FUNCTION_BLOCK AI_ChannelStatus
VAR
	{attribute addProperty Name  "<#Under Range#>"}
	UnderRange AT %I* : BIT;
	{attribute addProperty Name  "<#Over Range#>"}
	OverRange AT %I* : BIT;
	{attribute addProperty Name  "<#Value greater then limit 1#>"}
	Limit_1_Greater AT %I* : BIT;
	{attribute addProperty Name  "<#Value smaller then limit 1#>"}
	Limit_1_Smaller AT %I* : BIT;
	{attribute addProperty Name  "<#Value greater then limit 2#>"}
	Limit_2_Greater AT %I* : BIT;
	{attribute addProperty Name  "<#Value smaller then limit 2#>"}
	Limit_2_Smaller AT %I* : BIT;
	{attribute addProperty Name  "<#Error"}
	Error AT %I* : BIT;
	{attribute 'hide'}
	Reserved_1_7 AT %I* : BIT;
	{attribute 'hide'}
	Reserved_2_0 AT %I* : BIT;
	{attribute 'hide'}
	Reserved_2_1 AT %I* : BIT;
	{attribute 'hide'}
	Reserved_2_2 AT %I* : BIT;
	{attribute 'hide'}
	Reserved_2_3 AT %I* : BIT;
	{attribute 'hide'}
	Reserved_2_4 AT %I* : BIT;
	{attribute 'hide'}
	Reserved_2_5 AT %I* : BIT;
	{attribute addProperty Name  "<#TXPDO State#>"}
	TxPdoState AT %I* : BIT;
	{attribute addProperty Name  "<#TXPDO Toggle#>"}
	TxPdoToggle AT %I* : BIT;
END_VAR

END_FUNCTION_BLOCK

(* stored: Version 1.1.0.1, ProductVersion 3.1.4024.6
   POU AI_ChannelStatus: Id {4ba1bdec-761c-4800-b97a-c42a7cc8af14}, SpecialFunc None *)
